{attribute 'qualified_only'}
{attribute 'strict'}
TYPE E_NetworkByteOrder :
(
	BigEndian := 0, //Big Endian (MOTOROLA)
	LittleEndian := 1 //Little Endian (Intel)	
);
END_TYPE

(* stored: Version 1.1.0.1, ProductVersion 3.1.4024.12
   DUT E_NetworkByteOrder: Id {37325c95-aff9-083d-0d6e-6120f8b5dc6b} *)
